// TIA Portal project "CK_SCADA" (V16)

(* hardware
DEVICE "PC-System_1"  SIMATIC PC station
   slot 0: "SIMATIC PC station"  Rail  SIMATIC PC-Station  V1.0
      slot 125: "Stationmanager"  Station_Manager  V6.0.4
   slot 1: "HMI_RT_1"  WinCC RT Advanced  6AV2 104-0xxxx-xxxx  16.0.0.0
      slot 33792: "Computer interface"  Host interface
   slot 2: "IE general_1"  IE General  IE_CP  V8.2.0
DEVICE "S7-1200 station_1"  S7-1200 Station
   slot 0: "Rack_0"  S7-1200 Rack  Rack  V1.0
   slot 1: "PLC_1"  CPU 1215C AC/DC/Rly  6ES7 215-1BG40-0XB0  V4.4
   slot 101: "CM 1243-2"  CM 1243-2  3RK7243-2AA30-0XB0  V1.2
DEVICE "AS-i slave_1"  AS-i slave
   slot 0: "Rail_0"  Rail
   slot 1: "AS-i SM-I, 4DI_1"  AS-i SM-I, 4DI  3RK1 200-0CD00-0AA2
      slot 1: "AS-i SM-I, 4DI_1 [AS-i Slave (D)]"  AS-i Address-Module
      slot 2: "AS-i SM-I, 4DI_1 [AS-i Slave (A)]"  AS-i Address-Module
      slot 3: "AS-i SM-I, 4DI_1 [AS-i Slave (T)]"  AS-i Address-Module
DEVICE "AS-i slave_2"  AS-i slave
   slot 0: "Rail_0"  Rail
   slot 1: "AS-i SM-I, 4DI_2"  AS-i SM-I, 4DI  3RK1 200-0CD00-0AA2
      slot 1: "AS-i SM-I, 4DI_2 [AS-i Slave (D)]"  AS-i Address-Module
      slot 2: "AS-i SM-I, 4DI_2 [AS-i Slave (A)]"  AS-i Address-Module
      slot 3: "AS-i SM-I, 4DI_2 [AS-i Slave (T)]"  AS-i Address-Module
DEVICE "AS-i slave_3"  AS-i slave
   slot 0: "Rail_0"  Rail
   slot 1: "AS-i SM-I, 4DI_3"  AS-i SM-I, 4DI  3RK1 200-0CD00-0AA2
      slot 1: "AS-i SM-I, 4DI_3 [AS-i Slave (D)]"  AS-i Address-Module
      slot 2: "AS-i SM-I, 4DI_3 [AS-i Slave (A)]"  AS-i Address-Module
      slot 3: "AS-i SM-I, 4DI_3 [AS-i Slave (T)]"  AS-i Address-Module
DEVICE "AS-i slave_5"  AS-i slave
   slot 0: "Rail_0"  Rail
   slot 1: "AS-i SM-I, 4DI/4DO_1"  AS-i SM-I, 4DI/4DO  3RK1 400-1CD00-0AA2
      slot 1: "AS-i SM-I, 4DI/4DO_1 [AS-i Slave (D)]"  AS-i Address-Module
      slot 2: "AS-i SM-I, 4DI/4DO_1 [AS-i Slave (A)]"  AS-i Address-Module
      slot 3: "AS-i SM-I, 4DI/4DO_1 [AS-i Slave (T)]"  AS-i Address-Module
*)

// ===== PLC "PLC_1"  CPU 1215C AC/DC/Rly =====

VAR_GLOBAL   // PLC tag table "Default tag table"
   "System_Byte" AT %MB1 : Byte;
   "FirstScan" AT %M1.0 : Bool;
   "DiagStatusUpdate" AT %M1.1 : Bool;
   "AlwaysTRUE" AT %M1.2 : Bool;
   "AlwaysFALSE" AT %M1.3 : Bool;
   "System_Byte(1)" AT %MB1 : Byte;
   "Clock_Byte" AT %MB0 : Byte;
   "Clock_10Hz" AT %M0.0 : Bool;
   "Clock_5Hz" AT %M0.1 : Bool;
   "Clock_2.5Hz" AT %M0.2 : Bool;
   "Clock_2Hz" AT %M0.3 : Bool;
   "Clock_1.25Hz" AT %M0.4 : Bool;
   "Clock_1Hz" AT %M0.5 : Bool;
   "Clock_0.625Hz" AT %M0.6 : Bool;
   "Clock_0.5Hz" AT %M0.7 : Bool;
END_VAR

VAR_GLOBAL   // PLC tag table "input"
   "I_CALL_T1" AT %I2.0 : Bool;
   "I_CALL_T2_UP" AT %I2.1 : Bool;
   "I_CALL_T2_DW" AT %I2.2 : Bool;
   "I_CALL_T3" AT %I2.3 : Bool;
   "I_GH_DUOI" AT %I3.0 : Bool;
   "I_INSIDE_CALL_T1" AT %I3.1 : Bool;
   "I_INSIDE_CALL_T2" AT %I3.2 : Bool;
   "I_INSIDE_CALL_T3" AT %I3.3 : Bool;
   "I_DOOR_OPEN" AT %I4.0 : Bool;
   "I_DOOR_CLOSE" AT %I4.1 : Bool;
   "I_POSITION_T1" AT %I4.2 : Bool;
   "I_POSITION_T2" AT %I4.3 : Bool;
   "I_POSITION_T3" AT %I6.0 : Bool;
   "I_DOOR_OPENED" AT %I6.1 : Bool;
   "I_DOOR_CLOSED" AT %I6.2 : Bool;
END_VAR

VAR_GLOBAL   // PLC tag table "output"
   "Q_DOOR_OPEN" AT %Q2.0 : Bool;
   "Q_DOOR_CLOSE" AT %Q2.1 : Bool;
   "Q_BT_UP" AT %Q2.2 : Bool;
   "Q_BT_DW" AT %Q2.3 : Bool;
END_VAR

VAR_GLOBAL   // PLC tag table "TG"
   "NUT_SIMULATION" AT %M2.0 : Bool;
   "SI_POS_BT" AT %MW100 : Int;
   "SI_POS_DOOR" AT %MW102 : Int;
   "SI_POS_DOOR_T1" AT %MW104 : Int;
   "SI_POS_DOOR_T2" AT %MW106 : Int;
   "SI_POS_DOOR_T3" AT %MW108 : Int;
   "P1" AT %M30.0 : Bool;
   "P2" AT %M30.1 : Bool;
   "P3" AT %M30.2 : Bool;
   "P4" AT %M30.3 : Bool;
   "P5" AT %M30.4 : Bool;
   "P6" AT %M30.5 : Bool;
END_VAR

DATA_BLOCK "DATA_BUONGTHANG"   // DB1
{ S7_Optimized_Access := 'TRUE' }
VERSION : 0.1
// stored: InstanceOfName BUONG_DK
"BUONG_DK"
BEGIN
END_DATA_BLOCK

DATA_BLOCK "Data"   // DB3
{ S7_Optimized_Access := 'TRUE' }
VERSION : 0.1
   VAR
      HMI_DOOR_OPEN : Bool;
      HMI_DOOR_CLOSE : Bool;
      HMI_CALL_INSIDE_T1 : Bool;
      HMI_CALL_INSIDE_T2 : Bool;
      HMI_CALL_INSIDE_T3 : Bool;
      HMI_SHOW_INSIDE_T1 : Bool;
      HMI_SHOW_INSIDE_T2 : Bool;
      HMI_SHOW_INSIDE_T3 : Bool;
   END_VAR
BEGIN
END_DATA_BLOCK

// folder: System blocks/Program resources

DATA_BLOCK "IEC_Timer_0_DB"   // DB2
{ S7_Optimized_Access := 'TRUE' }
AUTHOR : Simatic
FAMILY : IEC
NAME : IEC_TMR
VERSION : 1.0
// stored: InstanceOfName IEC_TIMER
"IEC_TIMER"
BEGIN
END_DATA_BLOCK

// folder: (top level)

FUNCTION_BLOCK "BUONG_DK"   // FB1, LAD
{ S7_Optimized_Access := 'TRUE' }
VERSION : 0.1
   VAR_INPUT
      call_t1 : Bool;
      call_t2_up : Bool;
      call_t2_dw : Bool;
      call_t3 : Bool;
      pos_t1 : Bool;
      pos_t2 : Bool;
      pos_t3 : Bool;
      door_opened : Bool;
      door_closed : Bool;
      inside_t1 : Bool;
      inside_t2 : Bool;
      inside_t3 : Bool;
   END_VAR
   VAR_OUTPUT
      motor_up : Bool;
      motor_down : Bool;
   END_VAR
   VAR
      number_of_floor : Int;
      current_floor : Int;
      target_floor : Int;
      uping : Bool;
      downing : Bool;
      enable_scan_up : Bool;
      enable_scan_dw : Bool;
      scan_up_pos : Int;
      scan_dw_pos : Int;
      timer_reset_upping : IEC_TIMER;
      timer_reset_downing : IEC_TIMER;
      uu_tien_xep_hang_up : Array[0..4] of Bool;
      uu_tien_xep_hang_dw : Array[0..4] of Bool;
      dem_so_uu_tien_up : Int;
      dem_so_uu_tien_dw : Int;
      i : Int;
      j : Int;
   END_VAR
BEGIN

REGION Network 1 (SCL): thang máy có 3 tầng
   #number_of_floor := 3;
END_REGION

REGION Network 2 (SCL): gọi tầng ngoài buồng thang
   IF #call_t1 THEN
       #uu_tien_xep_hang_dw[1] := TRUE;
       #enable_scan_dw := TRUE;
   END_IF;
   //goi tang 2 di len
   IF #call_t2_up THEN
       #uu_tien_xep_hang_up[2] := TRUE;
       #enable_scan_up := TRUE;
   END_IF;
   //goi tang 2 di xuong 
   IF #call_t2_dw THEN
       #uu_tien_xep_hang_dw[2] := TRUE;
       #enable_scan_dw := TRUE;
   END_IF;
   //goi tang 2 di xuong 
   IF #call_t3 THEN
       #uu_tien_xep_hang_up[3] := TRUE;
       #enable_scan_up := TRUE;
   END_IF;
END_REGION

REGION Network 3 (SCL): Kiểm tra tầng hiện tại
   IF #pos_t1 THEN
       #current_floor := 1;
   END_IF;
   IF #pos_t2 THEN
       #current_floor := 2;
   END_IF;
   IF #pos_t3 THEN
       #current_floor := 3;
   END_IF;
END_REGION

REGION Network 4 (SCL): goi tang ben trong buong thang
   // Nếu thang ở tầng 1
   IF #current_floor = 1 THEN
       IF #inside_t2 THEN
           #uu_tien_xep_hang_up[2] := TRUE;
           #enable_scan_up := TRUE;
       END_IF;
       IF #inside_t3 THEN
           #uu_tien_xep_hang_up[3] := TRUE;
           #enable_scan_up := TRUE;
       END_IF;
   END_IF;
   IF #current_floor = 2 THEN
       IF #inside_t1 THEN
           #uu_tien_xep_hang_dw[1] := TRUE;
           #enable_scan_dw:= TRUE;
       END_IF;
       IF #inside_t3 THEN
           #uu_tien_xep_hang_up[3] := TRUE;
           #enable_scan_up := TRUE;
       END_IF;
   END_IF;
   IF #current_floor = 3 THEN
       IF #inside_t1 THEN
           #uu_tien_xep_hang_dw[1] := TRUE;
           #enable_scan_dw := TRUE;
       END_IF;
       IF #inside_t2 THEN
           #uu_tien_xep_hang_dw[2] := TRUE;
           #enable_scan_dw := TRUE;
       END_IF;
   END_IF;
END_REGION

REGION Network 5 (SCL): điều khiển di chuyển lên xuống dựa trên nút nhấn chọn tầng
   IF #current_floor < #target_floor AND #current_floor <> 0 THEN
       // Nếu tầng mục tiêu cao hơn, di chuyển lên
       IF #door_closed THEN // Chỉ di chuyển nếu cửa đã đóng hoàn toàn
           #motor_up := TRUE;
           #motor_down := FALSE;
       END_IF;

   ELSIF #current_floor > #target_floor THEN
       // Nếu tầng mục tiêu thấp hơn, di chuyển xuống
       IF #door_closed THEN // Chỉ di chuyển nếu cửa đã đóng hoàn toàn
           #motor_up := FALSE;
           #motor_down := TRUE;
       END_IF;

   ELSE
       // Nếu đã đến tầng mục tiêu, dừng động cơ
       #motor_up := FALSE;
       #motor_down := FALSE;
       // Loại bỏ yêu cầu từ hàng đợi
       IF #uping THEN
           #uu_tien_xep_hang_up[#current_floor] := FALSE;
       END_IF;

       IF #downing THEN
           #uu_tien_xep_hang_dw[#current_floor] := FALSE;
       END_IF;
   END_IF;
END_REGION

REGION Network 6 (SCL): Kiểm tra ưu tiên - đi lên

   IF #uping = FALSE THEN
       #scan_up_pos := 0;
   ELSE
       #scan_up_pos := #current_floor;

   END_IF;
      // Thang đi lên
   IF #enable_scan_up AND NOT #downing THEN
       #dem_so_uu_tien_up :=0;
       FOR #i := #current_floor TO #number_of_floor DO
           IF #uu_tien_xep_hang_up[#i] THEN
               #target_floor := #i;
               #uping := TRUE;
               #enable_scan_up := FALSE;
               #dem_so_uu_tien_up := #dem_so_uu_tien_up + 1;
               EXIT;
           END_IF;

           // Thoát vòng lặp khi chạy xong
           IF #i >= #number_of_floor AND #dem_so_uu_tien_up =0 THEN
               #enable_scan_up := FALSE;
               #uping := FALSE;
               EXIT;
           END_IF;
       END_FOR;
   END_IF;

   // Timer bật bit quét gọi tầng lên
   #timer_reset_upping.TON(IN := NOT #enable_scan_up,
                           PT := t#1s);

   IF #timer_reset_upping.Q = TRUE THEN
       #enable_scan_up := TRUE;
   END_IF;
END_REGION

REGION Network 7 (SCL): kiểm tra ưu tiên - đi xuống
   IF #downing = FALSE THEN
       #scan_dw_pos := 0;
   ELSE
       #scan_dw_pos := #current_floor;

   END_IF;
   // Thang đi xuong
   IF #enable_scan_dw AND NOT #uping THEN
       #dem_so_uu_tien_dw := 0;
       FOR #j := #current_floor TO 0 BY -1 DO
           IF #uu_tien_xep_hang_dw[#j] THEN
               #target_floor := #j;
               #downing := TRUE;
               #enable_scan_dw := FALSE;
               #dem_so_uu_tien_dw := #dem_so_uu_tien_dw + 1;
               EXIT;
           END_IF;

           // Thoát vòng lặp khi chạy xong
           IF #j = 0 AND #dem_so_uu_tien_dw =0 THEN
               #enable_scan_dw := FALSE;
               #downing := FALSE;
               EXIT;
           END_IF;
       END_FOR;
   END_IF;

   // Timer bật bit quét gọi tầng lên
   #timer_reset_downing.TON(IN := NOT #enable_scan_dw,
                           PT := t#1s);

   IF #timer_reset_downing.Q = TRUE THEN
       #enable_scan_dw := TRUE;
   END_IF;
END_REGION
END_FUNCTION_BLOCK

FUNCTION "CH_I_SANG_DB" : Void   // FC1, LAD
{ S7_Optimized_Access := 'TRUE' }
VERSION : 0.1
BEGIN

REGION Network 1 (SCL): nút gọi tầng
   "DATA_BUONGTHANG".call_t1 := "I_CALL_T1";
   "DATA_BUONGTHANG".call_t2_up := "I_CALL_T2_UP";
   "DATA_BUONGTHANG".call_t2_dw := "I_CALL_T2_DW";
   "DATA_BUONGTHANG".call_t3 := "I_CALL_T3";
END_REGION

REGION Network 2 (SCL): cảm biến
   "DATA_BUONGTHANG".pos_t1 := "I_POSITION_T1";
   "DATA_BUONGTHANG".pos_t2 := "I_POSITION_T2";
   "DATA_BUONGTHANG".pos_t3 := "I_POSITION_T3";
   "DATA_BUONGTHANG".door_closed := "I_DOOR_CLOSED";
   "DATA_BUONGTHANG".door_opened := "I_DOOR_OPENED";
END_REGION
END_FUNCTION

FUNCTION "DONG_MO_CUA" : Void   // FC2, LAD
{ S7_Optimized_Access := 'TRUE' }
VERSION : 0.1
   VAR_TEMP   // added for the SCL form of the ladder/FBD networks
      _w1 : Bool;
      _w2 : Bool;
   END_VAR
BEGIN

REGION Network 1: Reset cửa đóng khi cảm biến cửa đã đóng được tác động
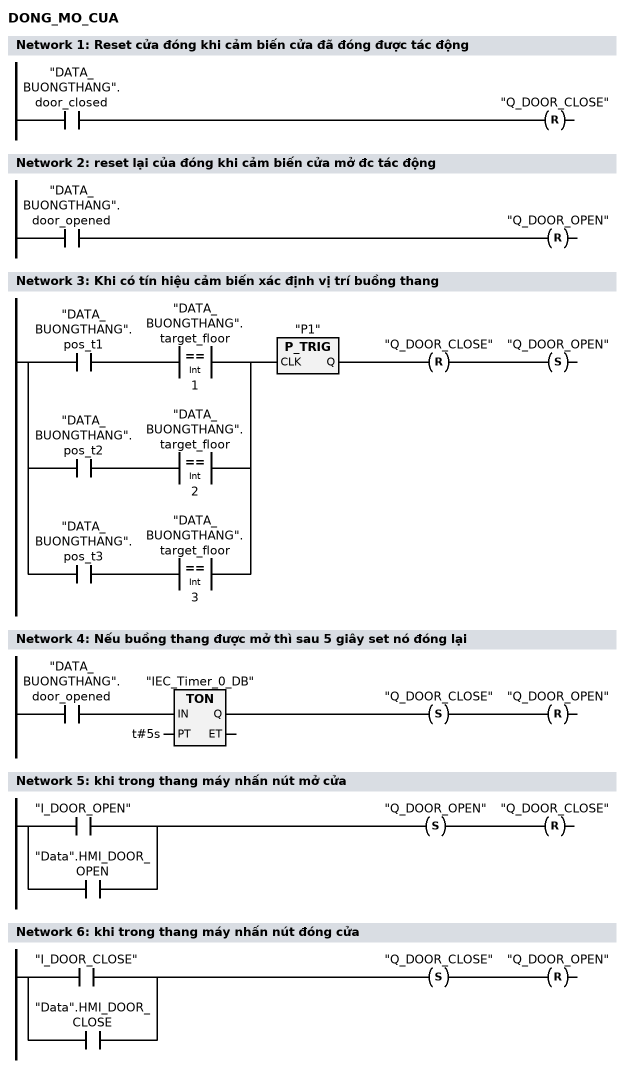
   RUNG wire#powerrail
      Contact( "DATA_BUONGTHANG".door_closed )
      R_Coil( "Q_DOOR_CLOSE" )
   END_RUNG
   // the same network as SCL:
   IF "DATA_BUONGTHANG".door_closed THEN "Q_DOOR_CLOSE" := FALSE; END_IF;
END_REGION

REGION Network 2: reset lại của đóng khi cảm biến cửa mở đc tác động
   RUNG wire#powerrail
      Contact( "DATA_BUONGTHANG".door_opened )
      R_Coil( "Q_DOOR_OPEN" )
   END_RUNG
   // the same network as SCL:
   IF "DATA_BUONGTHANG".door_opened THEN "Q_DOOR_OPEN" := FALSE; END_IF;
END_REGION

REGION Network 3: Khi có tín hiệu cảm biến xác định vị trí buồng thang
   RUNG wire#powerrail
      Contact( "DATA_BUONGTHANG".pos_t1 )
      { S7_Templates := "SrcType := Int" } EQ_Contact(in1 := "DATA_BUONGTHANG".target_floor, in2 := 1)
      wire#w1
      P_Trig( "P1" )
      R_Coil( "Q_DOOR_CLOSE" )
      S_Coil( "Q_DOOR_OPEN" )
   END_RUNG
   RUNG wire#powerrail
      Contact( "DATA_BUONGTHANG".pos_t2 )
      { S7_Templates := "SrcType := Int" } EQ_Contact(in1 := "DATA_BUONGTHANG".target_floor, in2 := 2)
   END_RUNG wire#w1
   RUNG wire#powerrail
      Contact( "DATA_BUONGTHANG".pos_t3 )
      { S7_Templates := "SrcType := Int" } EQ_Contact(in1 := "DATA_BUONGTHANG".target_floor, in2 := 3)
   END_RUNG wire#w1
   // the same network as SCL:
   #_w1 := ("DATA_BUONGTHANG".pos_t1 AND ("DATA_BUONGTHANG".target_floor = 1)) OR ("DATA_BUONGTHANG".pos_t2 AND ("DATA_BUONGTHANG".target_floor = 2)) OR ("DATA_BUONGTHANG".pos_t3 AND ("DATA_BUONGTHANG".target_floor = 3));
   #_w2 := #_w1 AND NOT "P1";   // rising edge
   "P1" := #_w1;
   IF #_w2 THEN
       "Q_DOOR_CLOSE" := FALSE;
       "Q_DOOR_OPEN" := TRUE;
   END_IF;
END_REGION

REGION Network 4: Nếu buồng thang được mở thì sau 5 giây set nó đóng lại
   "IEC_Timer_0_DB".TON(IN := "DATA_BUONGTHANG".door_opened, PT := t#5s);
   IF "IEC_Timer_0_DB".Q THEN
       "Q_DOOR_CLOSE" := TRUE;
       "Q_DOOR_OPEN" := FALSE;
   END_IF;
END_REGION

REGION Network 5: khi trong thang máy nhấn nút mở cửa
   RUNG wire#powerrail
      Contact( "I_DOOR_OPEN" )
      wire#w1
      S_Coil( "Q_DOOR_OPEN" )
      R_Coil( "Q_DOOR_CLOSE" )
   END_RUNG
   RUNG wire#powerrail
      Contact( "Data".HMI_DOOR_OPEN )
   END_RUNG wire#w1
   // the same network as SCL:
   IF "I_DOOR_OPEN" OR "Data".HMI_DOOR_OPEN THEN
       "Q_DOOR_OPEN" := TRUE;
       "Q_DOOR_CLOSE" := FALSE;
   END_IF;
END_REGION

REGION Network 6: khi trong thang máy nhấn nút đóng cửa
   RUNG wire#powerrail
      Contact( "I_DOOR_CLOSE" )
      wire#w1
      S_Coil( "Q_DOOR_CLOSE" )
      R_Coil( "Q_DOOR_OPEN" )
   END_RUNG
   RUNG wire#powerrail
      Contact( "Data".HMI_DOOR_CLOSE )
   END_RUNG wire#w1
   // the same network as SCL:
   IF "I_DOOR_CLOSE" OR "Data".HMI_DOOR_CLOSE THEN
       "Q_DOOR_CLOSE" := TRUE;
       "Q_DOOR_OPEN" := FALSE;
   END_IF;
END_REGION
END_FUNCTION

FUNCTION "MP" : Void   // FC3, LAD
{ S7_Optimized_Access := 'TRUE' }
VERSION : 0.1
   VAR_TEMP   // added for the SCL form of the ladder/FBD networks
      _w1 : Bool;
      _w2 : Bool;
      _w3 : Bool;
      _w4 : Bool;
   END_VAR
BEGIN

REGION Network 1: mô phỏng vị trí buồng thang
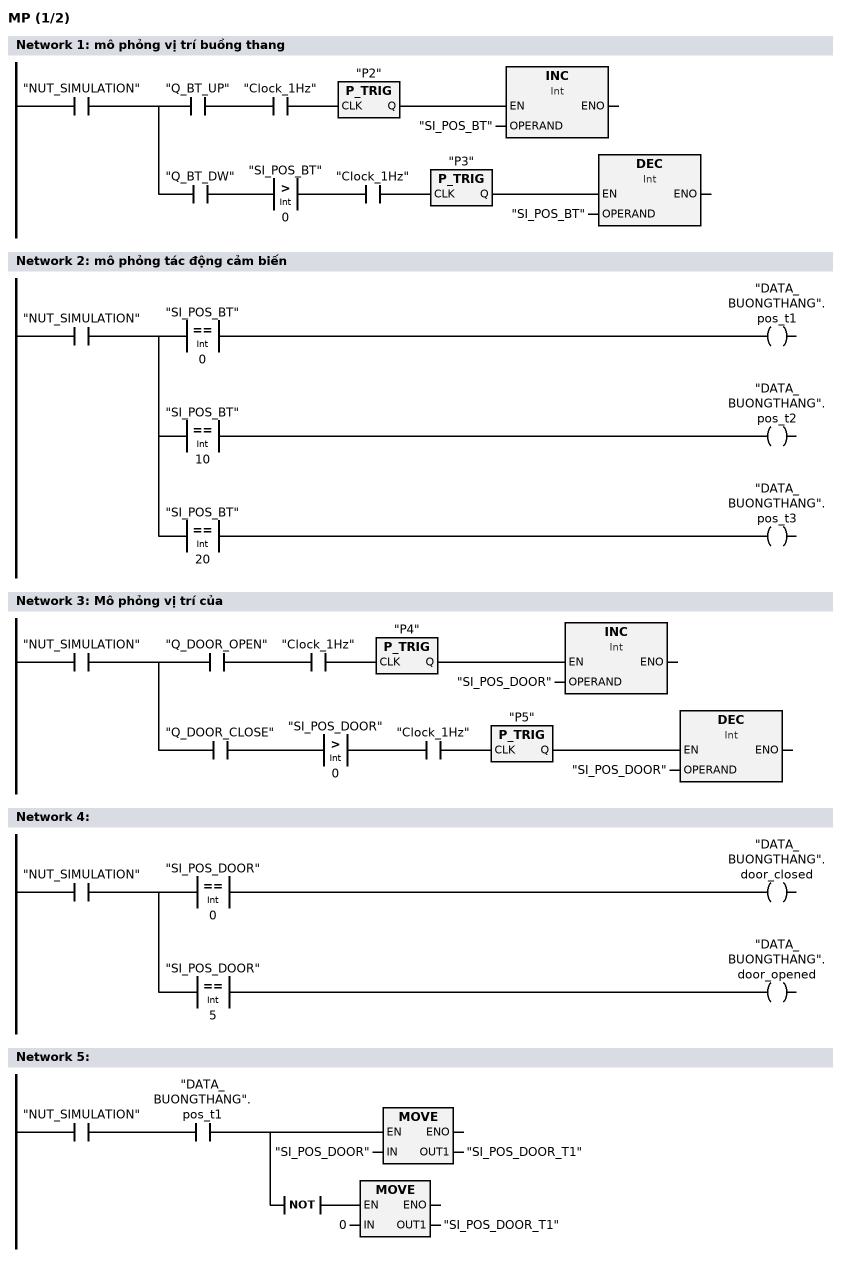
   RUNG wire#powerrail
      Contact( "NUT_SIMULATION" )
      wire#w1
      Contact( "Q_BT_UP" )
      Contact( "Clock_1Hz" )
      P_Trig( "P2" )
      { S7_Templates := "DestType := Int" } Inc( "SI_POS_BT" )
   END_RUNG
   RUNG wire#w1
      Contact( "Q_BT_DW" )
      { S7_Templates := "SrcType := Int" } GT_Contact(in1 := "SI_POS_BT", in2 := 0)
      Contact( "Clock_1Hz" )
      P_Trig( "P3" )
      { S7_Templates := "DestType := Int" } Dec( "SI_POS_BT" )
   END_RUNG
   // the same network as SCL:
   #_w1 := "NUT_SIMULATION" AND "Q_BT_UP" AND "Clock_1Hz";
   #_w2 := #_w1 AND NOT "P2";   // rising edge
   "P2" := #_w1;
   IF #_w2 THEN "SI_POS_BT" := "SI_POS_BT" + 1; END_IF;
   #_w3 := "NUT_SIMULATION" AND "Q_BT_DW" AND ("SI_POS_BT" > 0) AND "Clock_1Hz";
   #_w4 := #_w3 AND NOT "P3";   // rising edge
   "P3" := #_w3;
   IF #_w4 THEN "SI_POS_BT" := "SI_POS_BT" - 1; END_IF;
END_REGION

REGION Network 2: mô phỏng tác động cảm biến
   RUNG wire#powerrail
      Contact( "NUT_SIMULATION" )
      wire#w1
      { S7_Templates := "SrcType := Int" } EQ_Contact(in1 := "SI_POS_BT", in2 := 0)
      Coil( "DATA_BUONGTHANG".pos_t1 )
   END_RUNG
   RUNG wire#w1
      { S7_Templates := "SrcType := Int" } EQ_Contact(in1 := "SI_POS_BT", in2 := 10)
      Coil( "DATA_BUONGTHANG".pos_t2 )
   END_RUNG
   RUNG wire#w1
      { S7_Templates := "SrcType := Int" } EQ_Contact(in1 := "SI_POS_BT", in2 := 20)
      Coil( "DATA_BUONGTHANG".pos_t3 )
   END_RUNG
   // the same network as SCL:
   "DATA_BUONGTHANG".pos_t1 := "NUT_SIMULATION" AND ("SI_POS_BT" = 0);
   "DATA_BUONGTHANG".pos_t2 := "NUT_SIMULATION" AND ("SI_POS_BT" = 10);
   "DATA_BUONGTHANG".pos_t3 := "NUT_SIMULATION" AND ("SI_POS_BT" = 20);
END_REGION

REGION Network 3: Mô phỏng vị trí của
   RUNG wire#powerrail
      Contact( "NUT_SIMULATION" )
      wire#w1
      Contact( "Q_DOOR_OPEN" )
      Contact( "Clock_1Hz" )
      P_Trig( "P4" )
      { S7_Templates := "DestType := Int" } Inc( "SI_POS_DOOR" )
   END_RUNG
   RUNG wire#w1
      Contact( "Q_DOOR_CLOSE" )
      { S7_Templates := "SrcType := Int" } GT_Contact(in1 := "SI_POS_DOOR", in2 := 0)
      Contact( "Clock_1Hz" )
      P_Trig( "P5" )
      { S7_Templates := "DestType := Int" } Dec( "SI_POS_DOOR" )
   END_RUNG
   // the same network as SCL:
   #_w1 := "NUT_SIMULATION" AND "Q_DOOR_OPEN" AND "Clock_1Hz";
   #_w2 := #_w1 AND NOT "P4";   // rising edge
   "P4" := #_w1;
   IF #_w2 THEN "SI_POS_DOOR" := "SI_POS_DOOR" + 1; END_IF;
   #_w3 := "NUT_SIMULATION" AND "Q_DOOR_CLOSE" AND ("SI_POS_DOOR" > 0) AND "Clock_1Hz";
   #_w4 := #_w3 AND NOT "P5";   // rising edge
   "P5" := #_w3;
   IF #_w4 THEN "SI_POS_DOOR" := "SI_POS_DOOR" - 1; END_IF;
END_REGION

REGION Network 4
   RUNG wire#powerrail
      Contact( "NUT_SIMULATION" )
      wire#w1
      { S7_Templates := "SrcType := Int" } EQ_Contact(in1 := "SI_POS_DOOR", in2 := 0)
      Coil( "DATA_BUONGTHANG".door_closed )
   END_RUNG
   RUNG wire#w1
      { S7_Templates := "SrcType := Int" } EQ_Contact(in1 := "SI_POS_DOOR", in2 := 5)
      Coil( "DATA_BUONGTHANG".door_opened )
   END_RUNG
   // the same network as SCL:
   "DATA_BUONGTHANG".door_closed := "NUT_SIMULATION" AND ("SI_POS_DOOR" = 0);
   "DATA_BUONGTHANG".door_opened := "NUT_SIMULATION" AND ("SI_POS_DOOR" = 5);
END_REGION

REGION Network 5
   RUNG wire#powerrail
      Contact( "NUT_SIMULATION" )
      Contact( "DATA_BUONGTHANG".pos_t1 )
      wire#w1
      Move(in := "SI_POS_DOOR", out1 => "SI_POS_DOOR_T1")
   END_RUNG
   RUNG wire#w1
      Not()
      Move(in := 0, out1 => "SI_POS_DOOR_T1")
   END_RUNG
   // the same network as SCL:
   #_w1 := "NUT_SIMULATION" AND "DATA_BUONGTHANG".pos_t1;
   IF #_w1 THEN "SI_POS_DOOR_T1" := "SI_POS_DOOR"; END_IF;
   IF NOT #_w1 THEN "SI_POS_DOOR_T1" := 0; END_IF;
END_REGION

REGION Network 6
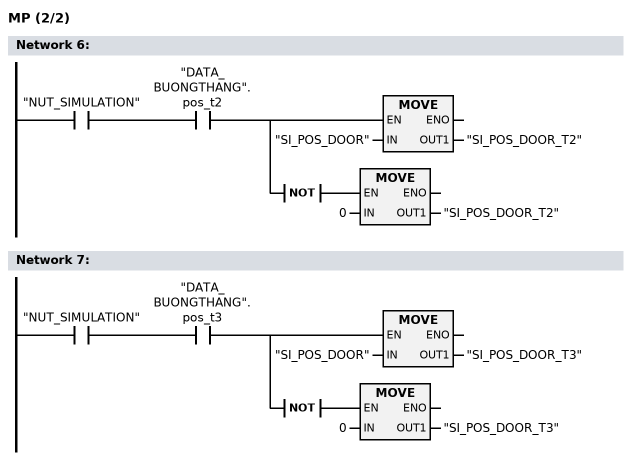
   RUNG wire#powerrail
      Contact( "NUT_SIMULATION" )
      Contact( "DATA_BUONGTHANG".pos_t2 )
      wire#w1
      Move(in := "SI_POS_DOOR", out1 => "SI_POS_DOOR_T2")
   END_RUNG
   RUNG wire#w1
      Not()
      Move(in := 0, out1 => "SI_POS_DOOR_T2")
   END_RUNG
   // the same network as SCL:
   #_w1 := "NUT_SIMULATION" AND "DATA_BUONGTHANG".pos_t2;
   IF #_w1 THEN "SI_POS_DOOR_T2" := "SI_POS_DOOR"; END_IF;
   IF NOT #_w1 THEN "SI_POS_DOOR_T2" := 0; END_IF;
END_REGION

REGION Network 7
   RUNG wire#powerrail
      Contact( "NUT_SIMULATION" )
      Contact( "DATA_BUONGTHANG".pos_t3 )
      wire#w1
      Move(in := "SI_POS_DOOR", out1 => "SI_POS_DOOR_T3")
   END_RUNG
   RUNG wire#w1
      Not()
      Move(in := 0, out1 => "SI_POS_DOOR_T3")
   END_RUNG
   // the same network as SCL:
   #_w1 := "NUT_SIMULATION" AND "DATA_BUONGTHANG".pos_t3;
   IF #_w1 THEN "SI_POS_DOOR_T3" := "SI_POS_DOOR"; END_IF;
   IF NOT #_w1 THEN "SI_POS_DOOR_T3" := 0; END_IF;
END_REGION
END_FUNCTION

FUNCTION "CALL_INSIDE" : Void   // FC4, LAD
{ S7_Optimized_Access := 'TRUE' }
VERSION : 0.1
BEGIN

REGION Network 1
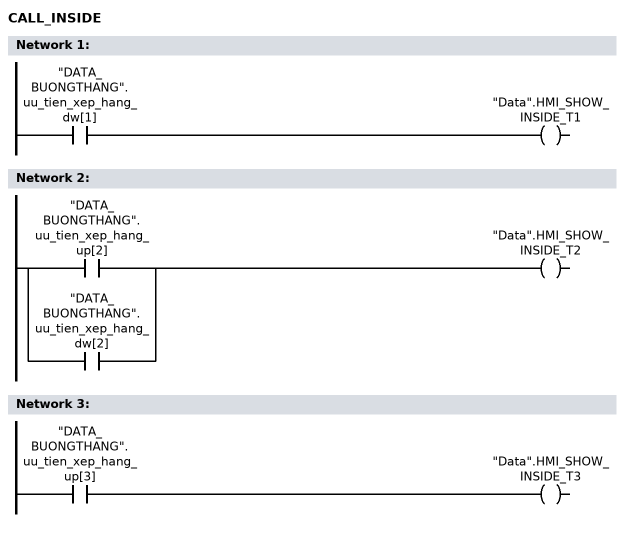
   RUNG wire#powerrail
      Contact( "DATA_BUONGTHANG".uu_tien_xep_hang_dw[1] )
      Coil( "Data".HMI_SHOW_INSIDE_T1 )
   END_RUNG
   // the same network as SCL:
   "Data".HMI_SHOW_INSIDE_T1 := "DATA_BUONGTHANG".uu_tien_xep_hang_dw[1];
END_REGION

REGION Network 2
   RUNG wire#powerrail
      Contact( "DATA_BUONGTHANG".uu_tien_xep_hang_up[2] )
      wire#w1
      Coil( "Data".HMI_SHOW_INSIDE_T2 )
   END_RUNG
   RUNG wire#powerrail
      Contact( "DATA_BUONGTHANG".uu_tien_xep_hang_dw[2] )
   END_RUNG wire#w1
   // the same network as SCL:
   "Data".HMI_SHOW_INSIDE_T2 := "DATA_BUONGTHANG".uu_tien_xep_hang_up[2] OR "DATA_BUONGTHANG".uu_tien_xep_hang_dw[2];
END_REGION

REGION Network 3
   RUNG wire#powerrail
      Contact( "DATA_BUONGTHANG".uu_tien_xep_hang_up[3] )
      Coil( "Data".HMI_SHOW_INSIDE_T3 )
   END_RUNG
   // the same network as SCL:
   "Data".HMI_SHOW_INSIDE_T3 := "DATA_BUONGTHANG".uu_tien_xep_hang_up[3];
END_REGION
END_FUNCTION

ORGANIZATION_BLOCK "Main"   // OB1, LAD, ProgramCycle
TITLE = "Main Program Sweep (Cycle)"
{ S7_Optimized_Access := 'TRUE' }
VERSION : 0.1
   VAR_INPUT
      Initial_Call : Bool;   // Initial call of this OB
      Remanence : Bool;   // =True, if remanent data are available
   END_VAR
BEGIN

REGION Network 1
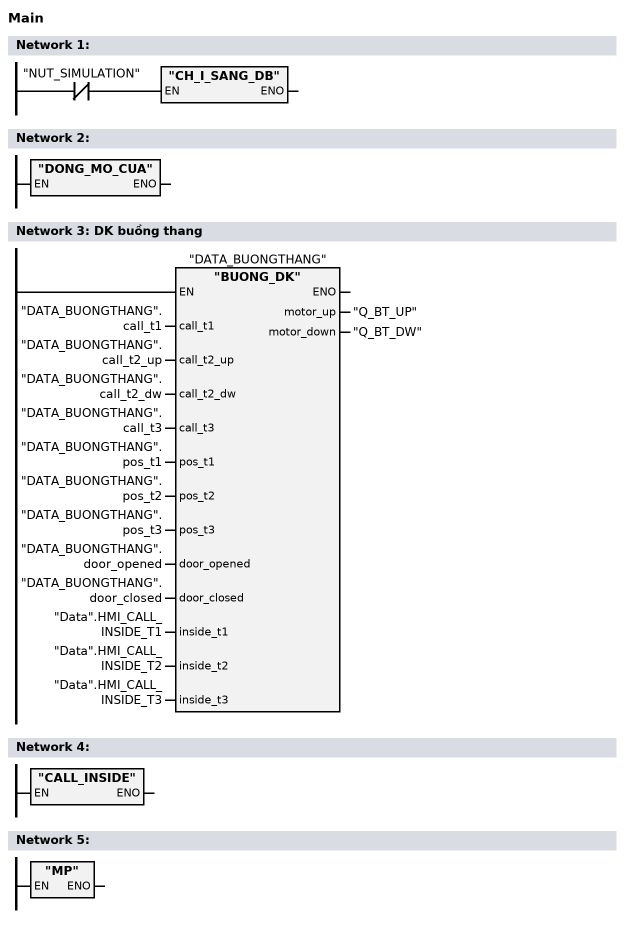
   RUNG wire#powerrail
      I_Contact( "NUT_SIMULATION" )
      "CH_I_SANG_DB"()
   END_RUNG
   // the same network as SCL:
   IF NOT "NUT_SIMULATION" THEN "CH_I_SANG_DB"(); END_IF;
END_REGION

REGION Network 2
   RUNG wire#powerrail
      "DONG_MO_CUA"()
   END_RUNG
   // the same network as SCL:
   "DONG_MO_CUA"();
END_REGION

REGION Network 3: DK buồng thang
   RUNG wire#powerrail
      "DATA_BUONGTHANG"(call_t1 := "DATA_BUONGTHANG".call_t1, call_t2_up := "DATA_BUONGTHANG".call_t2_up, call_t2_dw := "DATA_BUONGTHANG".call_t2_dw, call_t3 := "DATA_BUONGTHANG".call_t3, pos_t1 := "DATA_BUONGTHANG".pos_t1, pos_t2 := "DATA_BUONGTHANG".pos_t2, pos_t3 := "DATA_BUONGTHANG".pos_t3, door_opened := "DATA_BUONGTHANG".door_opened, door_closed := "DATA_BUONGTHANG".door_closed, inside_t1 := "Data".HMI_CALL_INSIDE_T1, inside_t2 := "Data".HMI_CALL_INSIDE_T2, inside_t3 := "Data".HMI_CALL_INSIDE_T3, motor_up => "Q_BT_UP", motor_down => "Q_BT_DW")
   END_RUNG
   // the same network as SCL:
   "DATA_BUONGTHANG"(call_t1 := "DATA_BUONGTHANG".call_t1,   // "BUONG_DK"
                     call_t2_up := "DATA_BUONGTHANG".call_t2_up,
                     call_t2_dw := "DATA_BUONGTHANG".call_t2_dw,
                     call_t3 := "DATA_BUONGTHANG".call_t3,
                     pos_t1 := "DATA_BUONGTHANG".pos_t1,
                     pos_t2 := "DATA_BUONGTHANG".pos_t2,
                     pos_t3 := "DATA_BUONGTHANG".pos_t3,
                     door_opened := "DATA_BUONGTHANG".door_opened,
                     door_closed := "DATA_BUONGTHANG".door_closed,
                     inside_t1 := "Data".HMI_CALL_INSIDE_T1,
                     inside_t2 := "Data".HMI_CALL_INSIDE_T2,
                     inside_t3 := "Data".HMI_CALL_INSIDE_T3,
                     motor_up => "Q_BT_UP",
                     motor_down => "Q_BT_DW");
END_REGION

REGION Network 4
   RUNG wire#powerrail
      "CALL_INSIDE"()
   END_RUNG
   // the same network as SCL:
   "CALL_INSIDE"();
END_REGION

REGION Network 5
   RUNG wire#powerrail
      "MP"()
   END_RUNG
   // the same network as SCL:
   "MP"();
END_REGION
END_ORGANIZATION_BLOCK

ORGANIZATION_BLOCK "Startup"   // OB100, LAD, Startup
TITLE = "Complete Restart"
{ S7_Optimized_Access := 'TRUE' }
VERSION : 0.1
   VAR_INPUT
      LostRetentive : Bool;   // True if retentive data are lost
      LostRTC : Bool;   // True if date and time are lost
   END_VAR
BEGIN

REGION Network 1
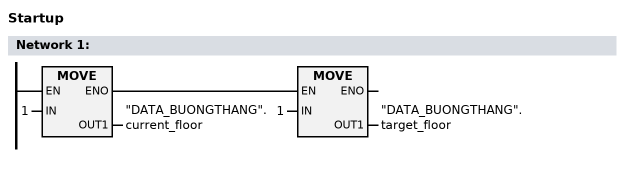
   RUNG wire#powerrail
      Move(in := 1, out1 => "DATA_BUONGTHANG".current_floor)
      Move(in := 1, out1 => "DATA_BUONGTHANG".target_floor)
   END_RUNG
   // the same network as SCL:
   "DATA_BUONGTHANG".current_floor := 1;
   "DATA_BUONGTHANG".target_floor := 1;
END_REGION
END_ORGANIZATION_BLOCK

(* ===== HMI "HMI_RT_1" =====
system functions are stored by id; their names below are inferred from use
connection "HMI_Connection_2": ETHERNET, S7_1200_OMS

HMI tags "Default tag table"
   "SI_POS_BT" : Int = PLC SI_POS_BT AT %MW100, 1 s
   "SI_POS_DOOR_T1" : Int = PLC SI_POS_DOOR_T1 AT %MW104, 1 s
   "SI_POS_DOOR_T2" : Int = PLC SI_POS_DOOR_T2 AT %MW106, 1 s
   "SI_POS_DOOR_T3" : Int = PLC SI_POS_DOOR_T3 AT %MW108, 1 s
   "DATA_BUONGTHANG_door_opened" : Bool = PLC DATA_BUONGTHANG.door_opened, 1 s
   "DATA_BUONGTHANG_door_closed" : Bool = PLC DATA_BUONGTHANG.door_closed, 1 s
   "DATA_BUONGTHANG_pos_t1" : Bool = PLC DATA_BUONGTHANG.pos_t1, 1 s
   "DATA_BUONGTHANG_call_t1" : Bool = PLC DATA_BUONGTHANG.call_t1, 1 s
   "DATA_BUONGTHANG_call_t3" : Bool = PLC DATA_BUONGTHANG.call_t3, 1 s
   "DATA_BUONGTHANG_call_t2_dw" : Bool = PLC DATA_BUONGTHANG.call_t2_dw, 1 s
   "DATA_BUONGTHANG_call_t2_up" : Bool = PLC DATA_BUONGTHANG.call_t2_up, 1 s
   "DATA_BUONGTHANG_uu_tien_xep_hang_dw{3}" : Bool = PLC DATA_BUONGTHANG.uu_tien_xep_hang_dw[3], 1 s
   "DATA_BUONGTHANG_uu_tien_xep_hang_dw{2}" : Bool = PLC DATA_BUONGTHANG.uu_tien_xep_hang_dw[2], 1 s
   "DATA_BUONGTHANG_uu_tien_xep_hang_up{1}" : Bool = PLC DATA_BUONGTHANG.uu_tien_xep_hang_up[1], 1 s
   "DATA_BUONGTHANG_uu_tien_xep_hang_up{2}" : Bool = PLC DATA_BUONGTHANG.uu_tien_xep_hang_up[2], 1 s
   "DATA_BUONGTHANG_uu_tien_xep_hang_dw{1}" : Bool = PLC DATA_BUONGTHANG.uu_tien_xep_hang_dw[1], 1 s
   "DATA_BUONGTHANG_uu_tien_xep_hang_up{3}" : Bool = PLC DATA_BUONGTHANG.uu_tien_xep_hang_up[3], 1 s
   "DATA_BUONGTHANG_current_floor" : Int = PLC DATA_BUONGTHANG.current_floor, 1 s
   "NUT_SIMULATION" : Bool = PLC NUT_SIMULATION AT %M2.0, 1 s
   "Data_HMI_DOOR_OPEN" : Bool = PLC Data.HMI_DOOR_OPEN, 1 s
   "Data_HMI_DOOR_CLOSE" : Bool = PLC Data.HMI_DOOR_CLOSE, 1 s
   "Data_HMI_CALL_INSIDE_T1" : Bool = PLC Data.HMI_CALL_INSIDE_T1, 1 s
   "Data_HMI_CALL_INSIDE_T2" : Bool = PLC Data.HMI_CALL_INSIDE_T2, 1 s
   "Data_HMI_CALL_INSIDE_T3" : Bool = PLC Data.HMI_CALL_INSIDE_T3, 1 s
   "Data_HMI_SHOW_INSIDE_T1" : Bool = PLC Data.HMI_SHOW_INSIDE_T1, 1 s
   "Data_HMI_SHOW_INSIDE_T2" : Bool = PLC Data.HMI_SHOW_INSIDE_T2, 1 s
   "Data_HMI_SHOW_INSIDE_T3" : Bool = PLC Data.HMI_SHOW_INSIDE_T3, 1 s
   "DATA_BUONGTHANG_pos_t2" : Bool = PLC DATA_BUONGTHANG.pos_t2, 1 s
   "DATA_BUONGTHANG_pos_t3" : Bool = PLC DATA_BUONGTHANG.pos_t3, 1 s

screen "Screen_1" 1024x768
   Rectangle "Rectangle_6" at 175,324 size 169x170
      HorizontalMovement <- "SI_POS_DOOR_T2"
   Rectangle "Rectangle_8" at 345,324 size 169x170
      HorizontalMovement <- "SI_POS_DOOR_T2"
   Rectangle "Rectangle_10" at 175,140 size 169x168
      HorizontalMovement <- "SI_POS_DOOR_T3"
   Rectangle "Rectangle_12" at 345,140 size 169x168
      HorizontalMovement <- "SI_POS_DOOR_T3"
   Rectangle "Rectangle_7" at 175,512 size 169x172
      HorizontalMovement <- "SI_POS_DOOR_T1"
   Rectangle "Rectangle_11" at 345,512 size 169x174
      HorizontalMovement <- "SI_POS_DOOR_T1"
   TextField "Text field_1" at 705,35 size 151x22; Text 'SCADA THANG MÁY'
   Rectangle "Rectangle_14" at 147,659 size 23x15
      Appearance <- "DATA_BUONGTHANG_pos_t1"
   Rectangle "Rectangle_15" at 146,496 size 23x15
      Appearance <- "DATA_BUONGTHANG_pos_t2"
   Rectangle "Rectangle_16" at 147,308 size 23x15
      Appearance <- "DATA_BUONGTHANG_pos_t3"
   Button "Button_1" at 669,144 size 60x32; TextOff '1'
      on Release: ResetBit("Data_HMI_CALL_INSIDE_T1")
      on Press: SetBit("Data_HMI_CALL_INSIDE_T1")
      Appearance <- "Data_HMI_SHOW_INSIDE_T1"
   Button "Button_2" at 841,145 size 58x32; TextOff '3'
      on Release: ResetBit("Data_HMI_CALL_INSIDE_T3")
      on Press: SetBit("Data_HMI_CALL_INSIDE_T3")
      Appearance <- "Data_HMI_SHOW_INSIDE_T3"
   Button "Button_3" at 753,144 size 60x32; TextOff '2'
      on Release: ResetBit("Data_HMI_CALL_INSIDE_T2")
      on Press: SetBit("Data_HMI_CALL_INSIDE_T2")
      Appearance <- "Data_HMI_SHOW_INSIDE_T2"
   Button "Button_4" at 698,258 size 76x32; TextOff 'ON'
      Appearance <- "NUT_SIMULATION"
      on Press: SetBit("NUT_SIMULATION")
   Button "Button_5" at 788,257 size 76x32; TextOff 'OFF'
      Appearance <- "NUT_SIMULATION"
      on Press: ResetBit("NUT_SIMULATION")
   TextField "Text field_2" at 701,235 size 161x22; Text 'Chức năng mô phỏng'
   Rectangle "Rectangle_24" at 26,516 size 96x162
      VerticalMovement <- "SI_POS_BT"
   Circle "Circle_1" at 625,366 size 42x42
      Appearance <- "DATA_BUONGTHANG_door_closed"
   Circle "Circle_2" at 625,417 size 42x42
      Appearance <- "DATA_BUONGTHANG_door_opened"
   Group "Group_3" at 523,202 size 34x36
   Group "Group_1" at 523,404 size 34x36
   Group "Group_2" at 523,597 size 34x36
   Group "Group_6" at 523,366 size 34x36
   IOField "I/O field_1" at 328,57 size 33x58; FormatPattern 9; Unit 0
      ProcessValue <- "DATA_BUONGTHANG_current_floor"
   IOField "I/O field_2" at 770,73 size 29x58; FormatPattern 9; Unit 0
      ProcessValue <- "DATA_BUONGTHANG_current_floor"
   Group "Group" at 708,188 size 66x34
   Group "Group_4" at 798,186 size 66x34
   TextField "Text field_3" at 686,371 size 152x34; Text 'CB cửa đóng'
   TextField "Text field_4" at 686,420 size 152x34; Text 'CB cửa mở'
   Button "Button_6" at 523,202 size 34x36; TextOff 'Text'
      on Press: SetBit("DATA_BUONGTHANG_call_t3")
      on Release: ResetBit("DATA_BUONGTHANG_call_t3")
      Appearance <- "DATA_BUONGTHANG_uu_tien_xep_hang_up{3}"
   Button "Button_7" at 523,404 size 34x36; TextOff 'Text'
      on Press: SetBit("DATA_BUONGTHANG_call_t2_dw")
      on Release: ResetBit("DATA_BUONGTHANG_call_t2_dw")
      Appearance <- "DATA_BUONGTHANG_uu_tien_xep_hang_dw{2}"
   Button "Button_8" at 523,597 size 34x36; TextOff 'Text'
      on Press: SetBit("DATA_BUONGTHANG_call_t1")
      on Release: ResetBit("DATA_BUONGTHANG_call_t1")
      Appearance <- "DATA_BUONGTHANG_uu_tien_xep_hang_dw{1}"
   Button "Button_9" at 523,366 size 34x36; TextOff 'Text'
      on Press: SetBit("DATA_BUONGTHANG_call_t2_up")
      on Release: ResetBit("DATA_BUONGTHANG_call_t2_up")
      Appearance <- "DATA_BUONGTHANG_uu_tien_xep_hang_up{2}"
   Button "Button_10" at 798,186 size 66x34; TextOff 'Text'
      on Release: ResetBit("Data_HMI_DOOR_CLOSE")
      on Press: SetBit("Data_HMI_DOOR_CLOSE")
      Appearance <- "Data_HMI_DOOR_CLOSE"
   Button "Button_11" at 708,188 size 66x34; TextOff 'Text'
      on Release: ResetBit("Data_HMI_DOOR_OPEN")
      on Press: SetBit("Data_HMI_DOOR_OPEN")
      Appearance <- "Data_HMI_DOOR_OPEN"
*)